SUBAPPLICATION Einstellungen (* Subapplication Type *)
  (* Standard: 61499-2 *)
  (* Version 1.0, 2024-04-23, Elias *)
  PACKAGE FBs::Baumsetzer::func::Einstellungen;
  IMPORT NVS_Keys::Key_Granulat_Dauer_Store;
  IMPORT NVS_Keys::Key_Granulatversatz_Store;
  IMPORT NVS_Keys::Key_Luft_Dauer_Store;
  IMPORT NVS_Keys::Key_Luftversatz_Store;
  IMPORT NVS_Keys::Key_Pflanzabstand_Store;
  IMPORT NVS_Keys::Key_Summer_Dauer_Store;
  IMPORT NVS_Keys::Key_Wasser_Dauer_Store;
  IMPORT NVS_Keys::Key_Wasserversatz_Store;
  IMPORT isobus::UT::io::Softkey::SoftKeyActivationCode::SK_RELEASED;
  IMPORT test::FBs::Baumsetzer::Constants::DefaultPool;
  IMPORT test::FBs::Baumsetzer::Constants::DefaultPool::SoftKey_Einstellungen;
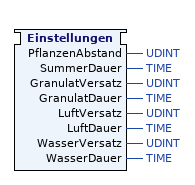
  VAR_OUTPUT
    PflanzenAbstand : UDINT := 12345; (* Pflanzabstand *)
    SummerDauer : TIME;
    GranulatVersatz : UDINT := 12345;
    GranulatDauer : TIME;
    LuftVersatz : UDINT := 12345;
    LuftDauer : TIME;
    WasserVersatz : UDINT := 12345;
    WasserDauer : TIME;
  END_VAR
  (* Group Reg_PflanzenAbstand: Einstellungen Pflanzabstand, per InputNumber *)
  (* Group Reg_Luftversatz: Einstellungen Pflanzabstand, per InputNumber *)
  (* Group Reg_Wasserversatz: Einstellungen Pflanzabstand, per InputNumber *)
  (* Group Reg_Granulatversatz: Einstellungen Pflanzabstand, per InputNumber *)
  (* Group Summer_Dauer: Einstellungen Pflanzabstand, per InputNumber *)
  (* Group Granulat_Dauer: Einstellungen Pflanzabstand, per InputNumber *)
  (* Group Luft_Dauer: Einstellungen Pflanzabstand, per InputNumber *)
  (* Group Wasser_Dauer: Einstellungen Pflanzabstand, per InputNumber *)
  FBS
    InputNumber_Pflanzabstand : isobus::UT::io::NumericValue::NumericValue_ID(QI := TRUE, u16ObjId := DefaultPool::InputNumber_Pflanzabstand); {SET_ATTRIBUTE(GroupName, Reg_PflanzenAbstand)}
    Q_NumericValue_Pflanzabstand : isobus::UT::Q::Q_NumericValue(u16ObjId := DefaultPool::InputNumber_Pflanzabstand); {SET_ATTRIBUTE(GroupName, Reg_PflanzenAbstand)}
    NVS_Pflanzabstand : logiBUS::storage::esp32_nvs::NVS(QI := TRUE, KEY := Key_Pflanzabstand_Store, DEFAULT_VALUE := UDINT#1000); {SET_ATTRIBUTE(GroupName, Reg_PflanzenAbstand)}
    F_DWORD_TO_UDINT_Pflanzabstand : iec61131::conversion::F_DWORD_TO_UDINT; {SET_ATTRIBUTE(GroupName, Reg_PflanzenAbstand)}
    InputNumber_Luftversatz : isobus::UT::io::NumericValue::NumericValue_ID(QI := TRUE, u16ObjId := DefaultPool::InputNumber_Luftversatz); {SET_ATTRIBUTE(GroupName, Reg_Luftversatz)}
    Q_NumericValue_Luftversatz : isobus::UT::Q::Q_NumericValue(u16ObjId := DefaultPool::InputNumber_Luftversatz); {SET_ATTRIBUTE(GroupName, Reg_Luftversatz)}
    NVS_Luftversatz : logiBUS::storage::esp32_nvs::NVS(QI := TRUE, KEY := Key_Luftversatz_Store, DEFAULT_VALUE := UDINT#1000); {SET_ATTRIBUTE(GroupName, Reg_Luftversatz)}
    F_DWORD_TO_UDINT_Luftversatz : iec61131::conversion::F_DWORD_TO_UDINT; {SET_ATTRIBUTE(GroupName, Reg_Luftversatz)}
    InputNumber_Wasserversatz : isobus::UT::io::NumericValue::NumericValue_ID(QI := TRUE, u16ObjId := DefaultPool::InputNumber_Wasserversatz); {SET_ATTRIBUTE(GroupName, Reg_Wasserversatz)}
    Q_NumericValue_Wasserversatz : isobus::UT::Q::Q_NumericValue(u16ObjId := DefaultPool::InputNumber_Wasserversatz); {SET_ATTRIBUTE(GroupName, Reg_Wasserversatz)}
    NVS_Wasserversatz : logiBUS::storage::esp32_nvs::NVS(QI := TRUE, KEY := Key_Wasserversatz_Store, DEFAULT_VALUE := UDINT#1000); {SET_ATTRIBUTE(GroupName, Reg_Wasserversatz)}
    F_DWORD_TO_UDINT_Wasserversatz : iec61131::conversion::F_DWORD_TO_UDINT; {SET_ATTRIBUTE(GroupName, Reg_Wasserversatz)}
    InputNumber_Granulatversatz : isobus::UT::io::NumericValue::NumericValue_ID(QI := TRUE, u16ObjId := DefaultPool::InputNumber_Granulatversatz); {SET_ATTRIBUTE(GroupName, Reg_Granulatversatz)}
    Q_NumericValue_Granulatversatz : isobus::UT::Q::Q_NumericValue(u16ObjId := DefaultPool::InputNumber_Granulatversatz); {SET_ATTRIBUTE(GroupName, Reg_Granulatversatz)}
    NVS_Granulatversatz : logiBUS::storage::esp32_nvs::NVS(QI := TRUE, KEY := Key_Granulatversatz_Store, DEFAULT_VALUE := UDINT#1000); {SET_ATTRIBUTE(GroupName, Reg_Granulatversatz)}
    F_DWORD_TO_UDINT_Granulatversatz : iec61131::conversion::F_DWORD_TO_UDINT; {SET_ATTRIBUTE(GroupName, Reg_Granulatversatz)}
    InputNumber_Summer_Dauer : isobus::UT::io::NumericValue::NumericValue_ID(QI := TRUE, u16ObjId := DefaultPool::InputNumber_Summer_Dauer); {SET_ATTRIBUTE(GroupName, Summer_Dauer)}
    Q_NumericValue_Summer_Dauer : isobus::UT::Q::Q_NumericValue(u16ObjId := DefaultPool::InputNumber_Summer_Dauer); {SET_ATTRIBUTE(GroupName, Summer_Dauer)}
    F_DWORD_TO_UDINT_Summer_Dauer : iec61131::conversion::F_DWORD_TO_UDINT; {SET_ATTRIBUTE(GroupName, Summer_Dauer)}
    NVS_Summer_Dauer : logiBUS::storage::esp32_nvs::NVS(QI := TRUE, KEY := Key_Summer_Dauer_Store, DEFAULT_VALUE := UDINT#1000); {SET_ATTRIBUTE(GroupName, Summer_Dauer)}
    InputNumber_Granulat_Dauer : isobus::UT::io::NumericValue::NumericValue_ID(QI := TRUE, u16ObjId := DefaultPool::InputNumber_Granulat_Dauer); {SET_ATTRIBUTE(GroupName, Granulat_Dauer)}
    Q_NumericValue_Granulat_Dauer : isobus::UT::Q::Q_NumericValue(u16ObjId := DefaultPool::InputNumber_Granulat_Dauer); {SET_ATTRIBUTE(GroupName, Granulat_Dauer)}
    F_DWORD_TO_UDINT_Granulat_Dauer : iec61131::conversion::F_DWORD_TO_UDINT; {SET_ATTRIBUTE(GroupName, Granulat_Dauer)}
    NVS_Granulat_Dauer : logiBUS::storage::esp32_nvs::NVS(QI := TRUE, KEY := Key_Granulat_Dauer_Store, DEFAULT_VALUE := UDINT#1000); {SET_ATTRIBUTE(GroupName, Granulat_Dauer)}
    InputNumber_Luft_Dauer : isobus::UT::io::NumericValue::NumericValue_ID(QI := TRUE, u16ObjId := DefaultPool::InputNumber_Luft_Dauer); {SET_ATTRIBUTE(GroupName, Luft_Dauer)}
    Q_NumericValue_Luft_Dauer : isobus::UT::Q::Q_NumericValue(u16ObjId := DefaultPool::InputNumber_Luft_Dauer); {SET_ATTRIBUTE(GroupName, Luft_Dauer)}
    F_DWORD_TO_UDINT_Luft_Dauer : iec61131::conversion::F_DWORD_TO_UDINT; {SET_ATTRIBUTE(GroupName, Luft_Dauer)}
    NVS_Luft_Dauer : logiBUS::storage::esp32_nvs::NVS(QI := TRUE, KEY := Key_Luft_Dauer_Store, DEFAULT_VALUE := UDINT#1000); {SET_ATTRIBUTE(GroupName, Luft_Dauer)}
    InputNumber_Wasser_Dauer : isobus::UT::io::NumericValue::NumericValue_ID(QI := TRUE, u16ObjId := DefaultPool::InputNumber_Wasser_Dauer); {SET_ATTRIBUTE(GroupName, Wasser_Dauer)}
    Q_NumericValue_Wasser_Dauer : isobus::UT::Q::Q_NumericValue(u16ObjId := DefaultPool::InputNumber_Wasser_Dauer); {SET_ATTRIBUTE(GroupName, Wasser_Dauer)}
    F_DWORD_TO_UDINT_Wasser_Dauer : iec61131::conversion::F_DWORD_TO_UDINT; {SET_ATTRIBUTE(GroupName, Wasser_Dauer)}
    NVS_Wasser_Dauer : logiBUS::storage::esp32_nvs::NVS(QI := TRUE, KEY := Key_Wasser_Dauer_Store, DEFAULT_VALUE := UDINT#1000); {SET_ATTRIBUTE(GroupName, Wasser_Dauer)}
    SoftKey_F4 : isobus::UT::io::Softkey::Softkey_IE(QI := TRUE, u16ObjId := SoftKey_Einstellungen, InputEvent := SK_RELEASED);
    F_MOVE : iec61131::selection::F_MOVE; {SET_ATTRIBUTE(DataType, UDINT)} {SET_ATTRIBUTE(GroupName, Reg_PflanzenAbstand)}
    F_MOVE_1 : iec61131::selection::F_MOVE; {SET_ATTRIBUTE(DataType, UDINT)} {SET_ATTRIBUTE(GroupName, Summer_Dauer)}
    F_MULTIME_3 : iec61131::arithmetic::F_MULTIME(IN1 := T#1ms); {SET_ATTRIBUTE(GroupName, Wasser_Dauer)}
    F_MULTIME : iec61131::arithmetic::F_MULTIME(IN1 := T#1ms); {SET_ATTRIBUTE(GroupName, Summer_Dauer)}
    F_MOVE_6 : iec61131::selection::F_MOVE; {SET_ATTRIBUTE(DataType, UDINT)} {SET_ATTRIBUTE(GroupName, Reg_Granulatversatz)}
    F_MOVE_7 : iec61131::selection::F_MOVE; {SET_ATTRIBUTE(DataType, UDINT)} {SET_ATTRIBUTE(GroupName, Luft_Dauer)}
    F_MOVE_8 : iec61131::selection::F_MOVE; {SET_ATTRIBUTE(DataType, UDINT)} {SET_ATTRIBUTE(GroupName, Granulat_Dauer)}
    F_MULTIME_2 : iec61131::arithmetic::F_MULTIME(IN1 := T#1ms); {SET_ATTRIBUTE(GroupName, Luft_Dauer)}
    F_MOVE_3 : iec61131::selection::F_MOVE; {SET_ATTRIBUTE(DataType, UDINT)} {SET_ATTRIBUTE(GroupName, Reg_Wasserversatz)}
    F_MULTIME_1 : iec61131::arithmetic::F_MULTIME(IN1 := T#1ms); {SET_ATTRIBUTE(GroupName, Granulat_Dauer)}
    F_MOVE_5 : iec61131::selection::F_MOVE; {SET_ATTRIBUTE(DataType, UDINT)} {SET_ATTRIBUTE(GroupName, Wasser_Dauer)}
    F_MOVE_2 : iec61131::selection::F_MOVE; {SET_ATTRIBUTE(DataType, UDINT)} {SET_ATTRIBUTE(GroupName, Reg_Luftversatz)}
  END_FBS
  EVENT_CONNECTIONS
    NVS_Luftversatz.GETO TO Q_NumericValue_Luftversatz.REQ;
    NVS_Wasserversatz.GETO TO Q_NumericValue_Wasserversatz.REQ;
    NVS_Granulatversatz.INITO TO Q_NumericValue_Granulatversatz.INIT;
    NVS_Granulatversatz.GETO TO Q_NumericValue_Granulatversatz.REQ;
    F_DWORD_TO_UDINT_Luftversatz.CNF TO NVS_Luftversatz.SET;
    F_DWORD_TO_UDINT_Wasserversatz.CNF TO NVS_Wasserversatz.SET;
    F_DWORD_TO_UDINT_Granulatversatz.CNF TO NVS_Granulatversatz.SET;
    InputNumber_Pflanzabstand.IND TO F_DWORD_TO_UDINT_Pflanzabstand.REQ;
    InputNumber_Luftversatz.IND TO F_DWORD_TO_UDINT_Luftversatz.REQ;
    InputNumber_Wasserversatz.IND TO F_DWORD_TO_UDINT_Wasserversatz.REQ;
    InputNumber_Granulatversatz.IND TO F_DWORD_TO_UDINT_Granulatversatz.REQ;
    F_DWORD_TO_UDINT_Pflanzabstand.CNF TO NVS_Pflanzabstand.SET;
    NVS_Pflanzabstand.INITO TO Q_NumericValue_Pflanzabstand.INIT;
    NVS_Pflanzabstand.GETO TO Q_NumericValue_Pflanzabstand.REQ;
    F_DWORD_TO_UDINT_Summer_Dauer.CNF TO NVS_Summer_Dauer.SET;
    NVS_Summer_Dauer.INITO TO Q_NumericValue_Summer_Dauer.INIT;
    InputNumber_Summer_Dauer.IND TO F_DWORD_TO_UDINT_Summer_Dauer.REQ;
    NVS_Summer_Dauer.GETO TO Q_NumericValue_Summer_Dauer.REQ;
    NVS_Granulat_Dauer.GETO TO Q_NumericValue_Granulat_Dauer.REQ;
    NVS_Granulat_Dauer.INITO TO Q_NumericValue_Granulat_Dauer.INIT;
    InputNumber_Granulat_Dauer.IND TO F_DWORD_TO_UDINT_Granulat_Dauer.REQ;
    F_DWORD_TO_UDINT_Granulat_Dauer.CNF TO NVS_Granulat_Dauer.SET;
    NVS_Luft_Dauer.GETO TO Q_NumericValue_Luft_Dauer.REQ;
    NVS_Luft_Dauer.INITO TO Q_NumericValue_Luft_Dauer.INIT;
    InputNumber_Luft_Dauer.IND TO F_DWORD_TO_UDINT_Luft_Dauer.REQ;
    F_DWORD_TO_UDINT_Luft_Dauer.CNF TO NVS_Luft_Dauer.SET;
    NVS_Wasser_Dauer.GETO TO Q_NumericValue_Wasser_Dauer.REQ;
    NVS_Wasser_Dauer.INITO TO Q_NumericValue_Wasser_Dauer.INIT;
    InputNumber_Wasser_Dauer.IND TO F_DWORD_TO_UDINT_Wasser_Dauer.REQ;
    F_DWORD_TO_UDINT_Wasser_Dauer.CNF TO NVS_Wasser_Dauer.SET;
    SoftKey_F4.IND TO Q_NumericValue_Pflanzabstand.REQ;
    SoftKey_F4.IND TO Q_NumericValue_Luftversatz.REQ;
    SoftKey_F4.IND TO Q_NumericValue_Wasserversatz.REQ;
    SoftKey_F4.IND TO Q_NumericValue_Granulatversatz.REQ;
    SoftKey_F4.IND TO Q_NumericValue_Wasser_Dauer.REQ;
    SoftKey_F4.IND TO Q_NumericValue_Summer_Dauer.REQ;
    SoftKey_F4.IND TO Q_NumericValue_Granulat_Dauer.REQ;
    SoftKey_F4.IND TO Q_NumericValue_Luft_Dauer.REQ;
    NVS_Summer_Dauer.INITO TO NVS_Summer_Dauer.GET;
    NVS_Granulat_Dauer.INITO TO NVS_Granulat_Dauer.GET;
    NVS_Luft_Dauer.INITO TO NVS_Luft_Dauer.GET;
    NVS_Wasser_Dauer.INITO TO NVS_Wasser_Dauer.GET;
    NVS_Granulatversatz.INITO TO NVS_Granulatversatz.GET;
    NVS_Wasserversatz.INITO TO NVS_Wasserversatz.GET;
    NVS_Luftversatz.INITO TO NVS_Luftversatz.GET;
    NVS_Pflanzabstand.INITO TO NVS_Pflanzabstand.GET;
    F_MOVE_8.CNF TO F_MULTIME_1.REQ;
    F_MOVE_5.CNF TO F_MULTIME_3.REQ;
    F_MOVE_1.CNF TO F_MULTIME.REQ;
    F_MOVE_7.CNF TO F_MULTIME_2.REQ;
    NVS_Pflanzabstand.SETO TO F_MOVE.REQ;
    NVS_Pflanzabstand.GETO TO F_MOVE.REQ;
    NVS_Luftversatz.SETO TO F_MOVE_2.REQ;
    NVS_Luftversatz.GETO TO F_MOVE_2.REQ;
    NVS_Wasserversatz.SETO TO F_MOVE_3.REQ;
    NVS_Wasserversatz.GETO TO F_MOVE_3.REQ;
    NVS_Granulatversatz.SETO TO F_MOVE_6.REQ;
    NVS_Granulatversatz.GETO TO F_MOVE_6.REQ;
    NVS_Wasser_Dauer.SETO TO F_MOVE_5.REQ;
    NVS_Wasser_Dauer.GETO TO F_MOVE_5.REQ;
    NVS_Luft_Dauer.SETO TO F_MOVE_7.REQ;
    NVS_Luft_Dauer.GETO TO F_MOVE_7.REQ;
    NVS_Granulat_Dauer.SETO TO F_MOVE_8.REQ;
    NVS_Granulat_Dauer.GETO TO F_MOVE_8.REQ;
    NVS_Summer_Dauer.SETO TO F_MOVE_1.REQ;
    NVS_Summer_Dauer.GETO TO F_MOVE_1.REQ;
  END_CONNECTIONS
  DATA_CONNECTIONS
    NVS_Luftversatz.VALUEO TO Q_NumericValue_Luftversatz.u32NewValue;
    NVS_Wasserversatz.VALUEO TO Q_NumericValue_Wasserversatz.u32NewValue;
    NVS_Granulatversatz.VALUEO TO Q_NumericValue_Granulatversatz.u32NewValue;
    F_DWORD_TO_UDINT_Luftversatz.OUT TO NVS_Luftversatz.VALUE;
    F_DWORD_TO_UDINT_Wasserversatz.OUT TO NVS_Wasserversatz.VALUE;
    F_DWORD_TO_UDINT_Granulatversatz.OUT TO NVS_Granulatversatz.VALUE;
    InputNumber_Pflanzabstand.IN TO F_DWORD_TO_UDINT_Pflanzabstand.IN;
    InputNumber_Luftversatz.IN TO F_DWORD_TO_UDINT_Luftversatz.IN;
    InputNumber_Wasserversatz.IN TO F_DWORD_TO_UDINT_Wasserversatz.IN;
    InputNumber_Granulatversatz.IN TO F_DWORD_TO_UDINT_Granulatversatz.IN;
    F_DWORD_TO_UDINT_Pflanzabstand.OUT TO NVS_Pflanzabstand.VALUE;
    NVS_Pflanzabstand.VALUEO TO Q_NumericValue_Pflanzabstand.u32NewValue;
    NVS_Summer_Dauer.VALUEO TO Q_NumericValue_Summer_Dauer.u32NewValue;
    InputNumber_Summer_Dauer.IN TO F_DWORD_TO_UDINT_Summer_Dauer.IN;
    F_DWORD_TO_UDINT_Summer_Dauer.OUT TO NVS_Summer_Dauer.VALUE;
    F_DWORD_TO_UDINT_Granulat_Dauer.OUT TO NVS_Granulat_Dauer.VALUE;
    InputNumber_Granulat_Dauer.IN TO F_DWORD_TO_UDINT_Granulat_Dauer.IN;
    NVS_Granulat_Dauer.VALUEO TO Q_NumericValue_Granulat_Dauer.u32NewValue;
    F_DWORD_TO_UDINT_Luft_Dauer.OUT TO NVS_Luft_Dauer.VALUE;
    InputNumber_Luft_Dauer.IN TO F_DWORD_TO_UDINT_Luft_Dauer.IN;
    NVS_Luft_Dauer.VALUEO TO Q_NumericValue_Luft_Dauer.u32NewValue;
    F_DWORD_TO_UDINT_Wasser_Dauer.OUT TO NVS_Wasser_Dauer.VALUE;
    InputNumber_Wasser_Dauer.IN TO F_DWORD_TO_UDINT_Wasser_Dauer.IN;
    NVS_Wasser_Dauer.VALUEO TO Q_NumericValue_Wasser_Dauer.u32NewValue;
    F_MOVE_5.OUT TO F_MULTIME_3.IN2;
    F_MOVE_8.OUT TO F_MULTIME_1.IN2;
    F_MOVE_7.OUT TO F_MULTIME_2.IN2;
    F_MOVE_1.OUT TO F_MULTIME.IN2;
    F_MOVE.OUT TO PflanzenAbstand;
    NVS_Pflanzabstand.VALUEO TO F_MOVE.IN;
    F_MULTIME.OUT TO SummerDauer;
    F_MOVE_6.OUT TO GranulatVersatz;
    F_MULTIME_1.OUT TO GranulatDauer;
    F_MOVE_2.OUT TO LuftVersatz;
    F_MULTIME_2.OUT TO LuftDauer;
    F_MOVE_3.OUT TO WasserVersatz;
    F_MULTIME_3.OUT TO WasserDauer;
    NVS_Granulatversatz.VALUEO TO F_MOVE_6.IN;
    NVS_Wasserversatz.VALUEO TO F_MOVE_3.IN;
    NVS_Luftversatz.VALUEO TO F_MOVE_2.IN;
    NVS_Wasser_Dauer.VALUEO TO F_MOVE_5.IN;
    NVS_Luft_Dauer.VALUEO TO F_MOVE_7.IN;
    NVS_Granulat_Dauer.VALUEO TO F_MOVE_8.IN;
    NVS_Summer_Dauer.VALUEO TO F_MOVE_1.IN;
  END_CONNECTIONS
END_SUBAPPLICATION
